{attribute 'GeneratedUsingTerminal: EL6201-0000-0017'}
{attribute addProperty BoxType "EL6201-0000-0017"}
{attribute addProperty Id "Slave_10A_DO0BOOL1Slave_10A_DO1BOOL1Slave_10A_DO2BOOL1Slave_10A_DO3BOOL1Slave_10B_DO0BOOL1Slave_10B_DO1BOOL1Slave_10B_DO2BOOL1Slave_10B_DO3BOOL1"}
{attribute addProperty CRC "267303882"}
{attribute addProperty Size "8"}
TYPE Slave_10_Outputs_0FEEBBCA :
STRUCT
	{attribute addProperty Name "Slave_10A_DO0"}
	Slave_10A_DO0 : BOOL;
	{attribute addProperty Name "Slave_10A_DO1"}
	Slave_10A_DO1 : BOOL;
	{attribute addProperty Name "Slave_10A_DO2"}
	Slave_10A_DO2 : BOOL;
	{attribute addProperty Name "Slave_10A_DO3"}
	Slave_10A_DO3 : BOOL;
	{attribute addProperty Name "Slave_10B_DO0"}
	Slave_10B_DO0 : BOOL;
	{attribute addProperty Name "Slave_10B_DO1"}
	Slave_10B_DO1 : BOOL;
	{attribute addProperty Name "Slave_10B_DO2"}
	Slave_10B_DO2 : BOOL;
	{attribute addProperty Name "Slave_10B_DO3"}
	Slave_10B_DO3 : BOOL;
END_STRUCT
END_TYPE

(* stored: Version 1.2.0.0, ProductVersion 3.1.4024.9
   DUT Slave_10_Outputs_0FEEBBCA: Id {4da9e116-8e67-4653-8cc1-f4c44d23f5b0} *)
